SUBAPPLICATION MSG_SUBSCRIBER (* ROS 2 MSG Subscriber *)
  (* Standard: 61499-2 *)
  (* Version 1.0, 2023-03-14, Tim Hesse *)
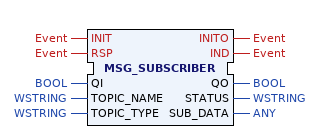
  EVENT_INPUT
    INIT; (* Initialization Request *)
    RSP; (* Application Response to IND *)
  END_EVENT
  EVENT_OUTPUT
    INITO; (* Initialization Confirm *)
    IND; (* Confirmation of Requested Service *)
  END_EVENT
  VAR_INPUT
    QI : BOOL; (* Input event qualifier *)
    TOPIC_NAME : WSTRING; (* ROS 2 Topic Name *)
    TOPIC_TYPE : WSTRING; (* ROS 2 Topic Type *)
  END_VAR
  VAR_OUTPUT
    QO : BOOL; (* Output event qualifier *)
    STATUS : WSTRING; (* Service Status *)
    SUB_DATA : ANY; (* Subscribed Data *)
  END_VAR
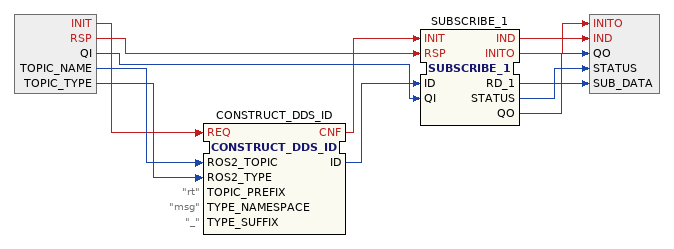
  FBS
    CONSTRUCT_DDS_ID : CONSTRUCT_DDS_ID(TOPIC_PREFIX := "rt", TYPE_NAMESPACE := "msg", TYPE_SUFFIX := "_");
    SUBSCRIBE_1 : SUBSCRIBE_1;
  END_FBS
  EVENT_CONNECTIONS
    INIT TO CONSTRUCT_DDS_ID.REQ;
    CONSTRUCT_DDS_ID.CNF TO SUBSCRIBE_1.INIT;
    RSP TO SUBSCRIBE_1.RSP;
    SUBSCRIBE_1.IND TO IND;
    SUBSCRIBE_1.INITO TO INITO;
  END_CONNECTIONS
  DATA_CONNECTIONS
    TOPIC_NAME TO CONSTRUCT_DDS_ID.ROS2_TOPIC;
    TOPIC_TYPE TO CONSTRUCT_DDS_ID.ROS2_TYPE;
    CONSTRUCT_DDS_ID.ID TO SUBSCRIBE_1.ID;
    QI TO SUBSCRIBE_1.QI;
    SUBSCRIBE_1.RD_1 TO SUB_DATA;
    SUBSCRIBE_1.STATUS TO STATUS;
    SUBSCRIBE_1.QO TO QO;
  END_CONNECTIONS
END_SUBAPPLICATION
